PROGRAM MAIN
VAR
	bRunOnlyOnce : BOOL := FALSE;
END_VAR

IF NOT bRunOnlyOnce THEN
	ADSLOGSTR(msgCtrlMask := ADSLOG_MSGTYPE_ERROR OR ADSLOG_MSGTYPE_LOG,
			  msgFmtStr := 'HelloWorld!',
			  strArg := '');
	bRunOnlyOnce := TRUE;
END_IF

END_PROGRAM

(* stored: Version 1.1.0.1, ProductVersion 3.1.4024.12
   POU MAIN: Id {8c21d7c9-0a50-4d3b-a8bc-ff8ef03f6452}, SpecialFunc None *)
